FUNCTION_BLOCK TcOpenTutorial EXTENDS TcoCore.TcoContext
VAR
	//101_Color_Sequencer
	ColorExample : Color_Example;
	
	//201 Connect sequencers
	ConnectSequences : ConnectSequences;
	
	//301 Invoking tasks
	InvokingTasks : InvokingTasks;
	//302 Task exectuion
	TaskExecution : TaskExecution;

END_VAR

// Use Main method instead of this block.

(*~
	<docu>
		<summary>
			Main method of the TcoContext. This is the entry point of any control logic that belongs to this context. 
			The call of this method is ensured by calling the <c>InstanceName.Run()</c> method, and it must not be called explicitly.
			This method is abstract, and it must be overridden in derived block.
		</summary>
	</docu>
~*)
METHOD PROTECTED  Main
ColorExample.Run();
ConnectSequences.Run();
InvokingTasks.Run();
TaskExecution.Run();
END_METHOD

END_FUNCTION_BLOCK

(* stored: Version 1.1.0.1, ProductVersion 3.1.4024.6
   POU TcOpenTutorial: Id {05284e7c-085c-0fc1-3da1-2c0f53b1a15c}, SpecialFunc None
   Method Main: Id {5e01554d-4a2b-0408-1aeb-e4bf0f739acc} *)
